(* CoDeSys 2.3 library: TIMER_ALARM.lib *)
(* Libraries: STANDARD.LIB 5.6.98 11:03:02 *)

(* POU MAIN, LD *)
PROGRAM MAIN
VAR
END_VAR
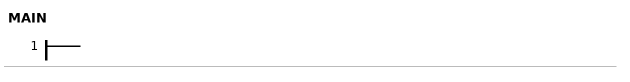
_LD_ (* Ladder Diagram *)
NETWORK 1
	*
_END_LD_
(* the same logic as Structured Text *)
(* Network 1 *)
END_PROGRAM

(* POU TIMER_ALARM, LD *)
FUNCTION_BLOCK TIMER_ALARM
VAR_INPUT
	BOOL_SIGNAL_IN: BOOL;
	BOOL_ALMRST_PB: BOOL;
	BOOL_BZRST_PB: BOOL;
	INT_PV: INT;

END_VAR

VAR_OUTPUT
	ALM_MSG_BOOL: BOOL;
	BZ_OUT_BOOL: BOOL;
	EV_INT: INT;
END_VAR

VAR
	T1: TON;
	M0: BOOL;
	M1: BOOL;
	D200: TIME;
	D202: INT;
END_VAR
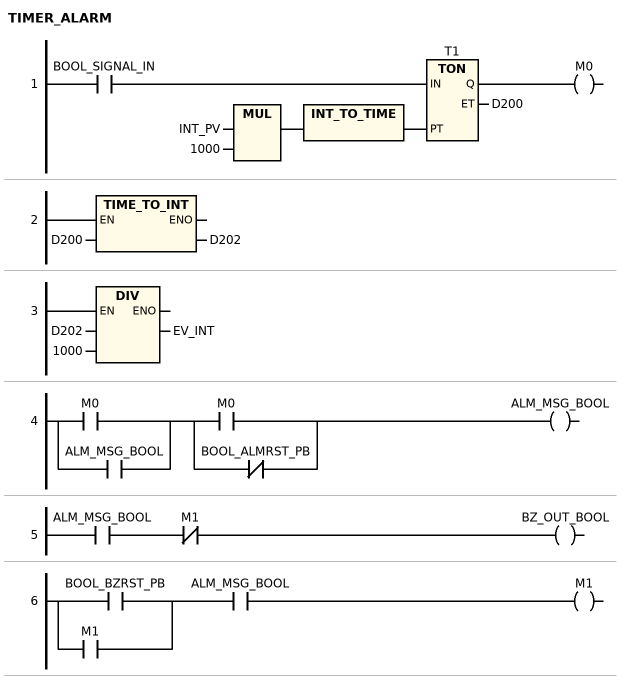
_LD_ (* Ladder Diagram *)
NETWORK 1
	[BOOL_SIGNAL_IN] - T1:TON(IN: *, PT: INT_TO_TIME(MUL(INT_PV, 1000)), ET => D200) --- (M0)
NETWORK 2
	*
		EN --- TIME_TO_INT(D200) => D202
NETWORK 3
	*
		EN --- DIV(D202, 1000) => EV_INT
NETWORK 4
	{ [M0] | [ALM_MSG_BOOL] } - { [M0] | [/BOOL_ALMRST_PB] } --- (ALM_MSG_BOOL)
NETWORK 5
	[ALM_MSG_BOOL] - [/M1] --- (BZ_OUT_BOOL)
NETWORK 6
	{ [BOOL_BZRST_PB] | [M1] } - [ALM_MSG_BOOL] --- (M1)
_END_LD_
(* the same logic as Structured Text *)
(* Network 1 *)
T1(IN := BOOL_SIGNAL_IN, PT := INT_TO_TIME(INT_PV * 1000));
D200 := T1.ET;
M0 := T1.Q;
(* Network 2 *)
D202 := TIME_TO_INT(D200);
(* Network 3 *)
EV_INT := D202 / 1000;
(* Network 4 *)
ALM_MSG_BOOL := ((M0) OR ALM_MSG_BOOL) AND (M0 OR NOT BOOL_ALMRST_PB);
(* Network 5 *)
BZ_OUT_BOOL := ALM_MSG_BOOL AND NOT M1;
(* Network 6 *)
M1 := (BOOL_BZRST_PB OR M1) AND ALM_MSG_BOOL;
END_FUNCTION_BLOCK
